% RSLogix 500 project timer.RSS, saved by version 8.30.00.16 %
PROJECT "UNTITLED"    % processor: Bul.1763 MicroLogix 1100 Series A %

PROGRAM FILES
  LAD 2   7 rungs

DATA FILES
  O0 OUTPUT  4 elements
  I1 INPUT  6 elements
  S2 STATUS  66 elements
  B3 BINARY  1 elements
  T4 TIMER  3 elements
  C5 COUNTER  2 elements
  R6 CONTROL  1 elements
  N7 INTEGER  1 elements
  F8 FLOAT  1 elements

LADDER 2
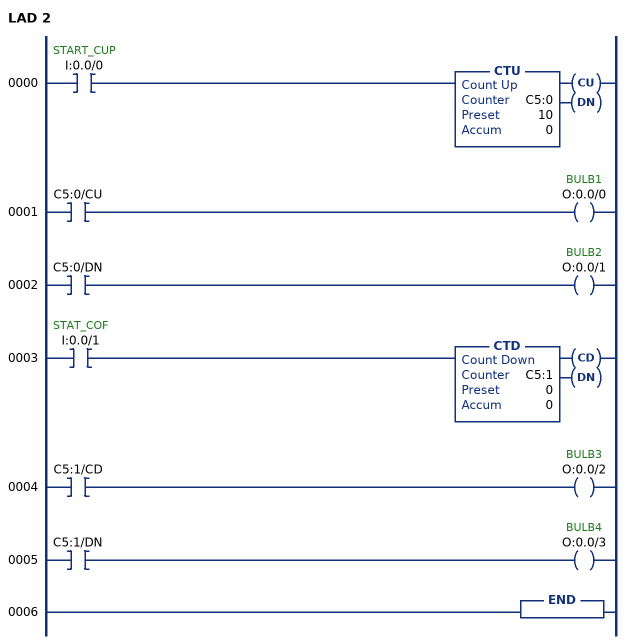
% Rung: 0 %
SOR XIC I:0.0/0 CTU C5:0 10 0 EOR
%   I:0.0/0  START_CUP %
% Rung: 1 %
SOR XIC C5:0/CU OTE O:0.0/0 EOR
%   O:0.0/0  BULB1 %
% Rung: 2 %
SOR XIC C5:0/DN OTE O:0.0/1 EOR
%   O:0.0/1  BULB2 %
% Rung: 3 %
SOR XIC I:0.0/1 CTD C5:1 0 0 EOR
%   I:0.0/1  STAT_COF %
% Rung: 4 %
SOR XIC C5:1/CD OTE O:0.0/2 EOR
%   O:0.0/2  BULB3 %
% Rung: 5 %
SOR XIC C5:1/DN OTE O:0.0/3 EOR
%   O:0.0/3  BULB4 %
% Rung: 6 %
SOR END EOR

OTHER DOCUMENTED ADDRESSES
  I:0.0/2  START_RTO
  I:0.0/3  BULB_4
  I:0.0/5  RESET
  O:0.0/4  BULB5
  O:0.0/5  BULB6

DATA TABLE (non-zero values as saved)
DATA T4
% .PRE .ACC %
% T4:0 % 20 0
% T4:1 % 10 10
% T4:2 % 30 0
DATA C5
% .PRE .ACC %
% C5:0 % 10 0
